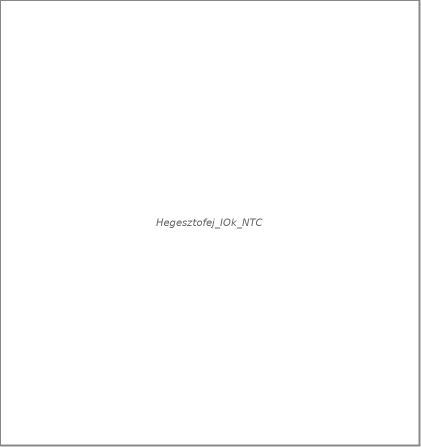
VISUALIZATION Hegesztofej_IOk  // 421x447
    TabControl (0,0 419x445), frame switch variable: GVL.iTengelyLapozo
        shows Hegesztofej_IOk_NTC()
        shows Hegesztofej_IOk_Pt()
        [0]: TabTitle=NTC oldal
        [1]: TabTitle=Pt oldal
END_VISUALIZATION

(* stored: Version 1.1.0.1, ProductVersion 3.1.4024.11
   Visu Hegesztofej_IOk: Id {adf4921b-9db8-4bc3-a98f-65c1420d19a2} *)
